(* IEC 61131-3 sources: LASAL/Class/SetCurrent, 1 file *)

(* ---- SetCurrent.st ---- *)
(*!
<Class
	Name               = "SetCurrent"
	Revision           = "0.0"
	RealtimeTask       = "false"
	CyclicTask         = "false"
	BackgroundTask     = "false"
	Sigmatek           = "false"
	OSInterface        = "false"
	HighPriority       = "false"
	Automatic          = "false"
	UpdateMode         = "Prescan"
	SharedCommandTable = "true"
	Objectsize         = "(284,120)">
	<Channels>
		<Server Name="ClassSvr" Visualized="false" Initialize="false" WriteProtected="true" Retentive="false"/>
		<Client Name="Current" Required="true" Internal="false"/>
	</Channels>
</Class>
*)
SetCurrent : CLASS
  //Servers:
	ClassSvr 	: SvrChCmd_DINT;
  //Clients:
	Current 	: CltCh_DINT;
  //Variables:
  //Functions:

	FUNCTION VIRTUAL GLOBAL Init;
  //Tables:
	FUNCTION @STD
		VAR_OUTPUT
			ret_code	: CONFSTATES;
		END_VAR;
	FUNCTION GLOBAL TAB @CT_;
END_CLASS;

FUNCTION VIRTUAL GLOBAL SetCurrent::Init
Current.Write(input:=1000);
END_FUNCTION
